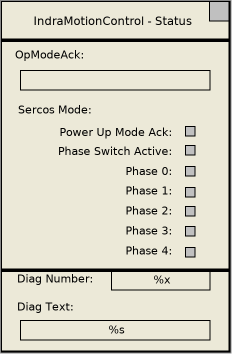
VISUALIZATION ImcStatus  // 232x354
    Rectangle (0,0 230x352)
    Rectangle (13,11 200x20), "IndraMotionControl - Status"
    Rectangle (209,1 20x20), colour toggle: Global_ImcInterface.ImcStatus .InOperation
    Rectangle (12,45 96x20), "OpModeAck:"
    Rectangle (20,70 190x20), text list: 'ImcModeStatus', text index: Global_ImcInterface.ImcStatus .Admin._OpModeAck
    Rectangle (0,40 230x0)
    Rectangle (15,100 90x20), "Sercos Mode:"
    Rectangle (0,270 230x0)
    Rectangle (185,187 10x10), colour toggle: Global_ImcInterface.ImcStatus .Admin.ModeStatus_P1
    Rectangle (185,226 10x10), colour toggle: Global_ImcInterface.ImcStatus .Admin.ModeStatus_P3
    Rectangle (185,206 10x10), colour toggle: Global_ImcInterface.ImcStatus .Admin.ModeStatus_P2
    Rectangle (185,166 10x10), colour toggle: Global_ImcInterface.ImcStatus .Admin.ModeStatus_P0
    Rectangle (185,247 10x10), colour toggle: Global_ImcInterface.ImcStatus .Admin.ModeStatus_BB
    Rectangle (185,145 10x10), colour toggle: Global_ImcInterface.ImcStatus .Admin.PhaseSwitchActive
    Rectangle (115,161 60x21), "Phase 0:"
    Rectangle (115,181 60x20), "Phase 1:"
    Rectangle (115,201 60x20), "Phase 2:"
    Rectangle (115,221 60x20), "Phase 3:"
    Rectangle (115,241 60x20), "Phase 4:"
    Rectangle (45,141 130x21), "Phase Switch Active:"
    Rectangle (45,125 130x15), "Power Up Mode Ack:"
    Rectangle (185,126 10x10), colour toggle: Global_ImcInterface.ImcStatus .Admin.PwrUpModeAck
    Rectangle (111,270 99x20), "%x", text variable: Global_ImcInterface.ImcStatus .Diag.Number
    Rectangle (20,320 190x20), "%s", text variable: Global_ImcInterface.ImcStatus .Diag.Message
    Rectangle (14,269 100x20), "Diag Number:"
    Rectangle (14,297 100x20), "Diag Text:"
END_VISUALIZATION

// IndraMotionMlc1/Application/AxisInterface/Visualizations/SystemOverview/System_Overview
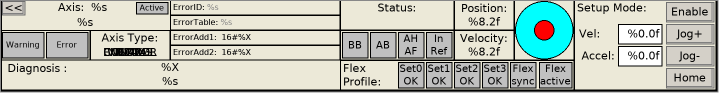
VISUALIZATION System_Overview  // 719x93
VAR_INPUT
	m_Input_AxisName : AXIS_REF;
END_VAR
    Rectangle (0,-1 717x92)
    Rectangle (1,61 340x15), "Diagnosis :"
    Rectangle (0,30 90x30)
    Rectangle (0,15 170x15), "%s", text variable: arAxisStatus_gb[m_Input_AxisName.AxisNo].Admin.Name
    Rectangle (340,30 114x30)
    Rectangle (514,0 60x60)
    Rectangle (24,0 117x15), "Axis: %s", text variable: m_Input_AxisName.AxisNo
    Rectangle (340,0 114x30), "Status:"
    Rectangle (454,0 60x30), "Position: %8.2f", text variable: AxisData[m_Input_AxisName.AxisNo].rActualPosition_i
    Rectangle (454,30 60x30), "Velocity: %8.2f", text variable: AxisData[m_Input_AxisName.AxisNo].rActualVelocity_i
    RoundedRectangle (342,32 26x26), "BB", colour toggle: (AxisData[m_Input_AxisName.Axisno].Axis_Inbb) <> 0
    RoundedRectangle (370,32 26x26), "AB", colour toggle: (AxisData[m_Input_AxisName.Axisno].Axis_InAb) <> 0
    RoundedRectangle (426,32 26x26), "In Ref", colour toggle: (AxisData[m_Input_AxisName.Axisno].Axis_Homed) <> 0
    RoundedRectangle (2,32 42x26), "Warning", colour toggle: (arAxisStatus_gb[m_Input_AxisName.Axisno].Diag.Warning) <> 0
    RoundedRectangle (46,32 42x26), "Error", colour toggle: (arAxisStatus_gb[m_Input_AxisName.Axisno].Diag.Error) <> 0
    RoundedRectangle (398,32 26x26), "AH AF", colour toggle: (AxisData[m_Input_AxisName.Axisno].Axis_Power) <> 0
    Ellipse (515,1 58x58)
    Polygon (0,0 0x0)
        p2858320360: AxisData[m_Input_AxisName.Axisno].rActualPosition_i
    Ellipse (534,20 20x20), colour toggle: (arAxisStatus_gb[m_Input_AxisName.AxisNo].Admin.Active) <> 0
    Rectangle (90,30 80x30), "Axis Type:"
    Rectangle (574,0 143x90), "Setup Mode:"
    Button (666,2 48x20), "Enable", colour toggle: arAxisStatus_gb[m_Input_AxisName.AxisNo].SetupMode.EnableAck, pressed state: arAxisCtrl_gb [m_Input_AxisName.AxisNo].SetupMode.Enable, input disabled if: bRemoteOn_gb = FALSE
        toggle arAxisCtrl_gb [m_Input_AxisName.AxisNo].SetupMode.Enable
    Button (666,24 48x20), "Jog+", input disabled if: (arAxisStatus_gb[m_Input_AxisName.AxisNo].SetupMode.EnableAck) = 0
        tap arAxisCtrl_gb [m_Input_AxisName.AxisNo].SetupMode.JogPlus
    Button (666,46 48x20), "Jog-", input disabled if: (arAxisStatus_gb[m_Input_AxisName.AxisNo].SetupMode.EnableAck) = 0
        tap arAxisCtrl_gb [m_Input_AxisName.AxisNo].SetupMode.JogMinus
    Button (666,68 48x20), "Home", colour toggle: arAxisStatus_gb[m_Input_AxisName.AxisNo].SetupMode.HomingAck, input disabled if: (arAxisStatus_gb[m_Input_AxisName.AxisNo].SetupMode.EnableAck) = 0
        tap arAxisCtrl_gb [m_Input_AxisName.AxisNo].SetupMode.Homing
    Rectangle (618,24 44x20), "%0.0f", text variable: arAxisCtrl_gb[m_Input_AxisName.AxisNo].SetupMode.Vel
        OnMouseUp: write arAxisCtrl_gb [m_Input_AxisName.AxisNo].SetupMode.Vel via Edit
    Rectangle (575,24 29x20), "Vel:"
    Rectangle (618,46 44x20), "%0.0f", text variable: arAxisCtrl_gb[m_Input_AxisName.AxisNo].SetupMode.Accel
        OnMouseUp: write arAxisCtrl_gb [m_Input_AxisName.AxisNo].SetupMode.Accel via Edit
    Rectangle (575,46 46x20), "Accel:"
    Button (2,1 23x14), "<<"
        OnMouseClick:  Assign=Axis_Overview, Type=Assignment
        OnMouseClick: execute { VisuAxisNo :=(m_Input_AxisName.AxisNo); }
    RoundedRectangle (136,2 32x12), "Active", colour toggle: (arAxisStatus_gb[m_Input_AxisName.AxisNo].Admin.Active) <> 0
    Rectangle (0,60 340x15), "%X", text variable: arAxisStatus_gb [m_Input_AxisName.AxisNo].Diag.Number, invisible if: arAxisStatus_gb [m_Input_AxisName.AxisNo].Diag.Number = 0
    RoundedRectangle (398,62 26x26), "Set0 OK", colour toggle: (AxisData[m_Input_AxisName.Axisno].FlexProfil_Set0_Ok) <> 0
    RoundedRectangle (426,62 26x26), "Set1 OK", colour toggle: (AxisData[m_Input_AxisName.Axisno].FlexProfil_Set1_Ok) <> 0
    RoundedRectangle (454,62 26x26), "Set2 OK", colour toggle: (AxisData[m_Input_AxisName.Axisno].FlexProfil_Set2_Ok) <> 0
    RoundedRectangle (482,62 26x26), "Set3 OK", colour toggle: (AxisData[m_Input_AxisName.Axisno].FlexProfil_Set3_Ok) <> 0
    Group (90,45 80x15)
        Rectangle (0,0 80x15), "REAL", invisible if: arAxisStatus_gb [m_Input_AxisName.AxisNo].Admin.AxisType <> RealAxisCfg
        Rectangle (0,0 80x15), "VIRTUAL", invisible if: arAxisStatus_gb [m_Input_AxisName.AxisNo].Admin.AxisType <> VirtualAxisCfg
        Rectangle (0,0 80x15), "ENCODER", invisible if: arAxisStatus_gb [m_Input_AxisName.AxisNo].Admin.AxisType <> EncoderAxisCfg
        Rectangle (0,0 80x15), "LINK", invisible if: arAxisStatus_gb [m_Input_AxisName.AxisNo].Admin.AxisType <> LinkAxisCfg
        Rectangle (0,0 80x15), "NO AXIS", invisible if: .arAxisStatus_gb [m_Input_AxisName.AxisNo].Admin.AxisType <> NoAxisConfig
        Rectangle (0,0 80x15), "CONTROL", invisible if: arAxisStatus_gb [m_Input_AxisName.AxisNo].Admin.AxisType <> ControlAxisCfg
    Rectangle (0,74 340x15), "%s", text variable: arAxisStatus_gb [m_Input_AxisName.AxisNo].Diag.Message
    Rectangle (170,0 170x15), "ErrorID: %s", text variable: arAxisStatus_gb [m_Input_AxisName.AxisNo].Diag.ErrorID, invisible if: (arAxisStatus_gb[m_Input_AxisName.Axisno].Diag.Error) <> 0
    Rectangle (170,0 170x15), "ErrorID:", invisible if: (arAxisStatus_gb[m_Input_AxisName.Axisno].Diag.Error) = 0, text list: 'ErrorIDCode', text index: arAxisStatus_gb [m_Input_AxisName.AxisNo].Diag.ErrorID
    Rectangle (170,15 170x15), "ErrorTable: %s", text variable: arAxisStatus_gb [m_Input_AxisName.AxisNo].Diag.ErrorIdent.Table, invisible if: (arAxisStatus_gb[m_Input_AxisName.Axisno].Diag.Error) <> 0
    Rectangle (170,15 170x15), "ErrorTable:", invisible if: (arAxisStatus_gb[m_Input_AxisName.Axisno].Diag.Error) = 0, text list: 'ErrorTable', text index: arAxisStatus_gb [m_Input_AxisName.AxisNo].Diag.ErrorIdent.Table
    Group (170,30 170x15)
        Rectangle (0,0 170x15), "ErrorAdd1: 16#%X", text variable: arAxisStatus_gb [m_Input_AxisName.AxisNo].Diag.ErrorIdent.Additional1, invisible if: (arAxisStatus_gb[m_Input_AxisName.Axisno].Diag.Error) <> 0
        Rectangle (0,0 170x15), "ErrorAdd1: 16#%X", text variable: arAxisStatus_gb [m_Input_AxisName.AxisNo].Diag.ErrorIdent.Additional1, invisible if: (arAxisStatus_gb[m_Input_AxisName.Axisno].Diag.Error) = 0
    Group (170,45 170x15)
        Rectangle (0,0 170x15), "ErrorAdd2: 16#%X", text variable: arAxisStatus_gb [m_Input_AxisName.AxisNo].Diag.ErrorIdent.Additional2, invisible if: (arAxisStatus_gb[m_Input_AxisName.Axisno].Diag.Error) <> 0
        Rectangle (0,0 170x15), "ErrorAdd2: 16#%X", text variable: arAxisStatus_gb [m_Input_AxisName.AxisNo].Diag.ErrorIdent.Additional2, invisible if: (arAxisStatus_gb[m_Input_AxisName.Axisno].Diag.Error) = 0
    Rectangle (340,60 234x30), "Flex Profile:"
    RoundedRectangle (539,62 33x26), "Flex active", colour toggle: (AxisData[m_Input_AxisName.Axisno].FlexProfil_Active) <> 0
    RoundedRectangle (510,62 26x26), "Flex sync", colour toggle: (AxisData[m_Input_AxisName.Axisno].FlexProfil_Sync) <> 0
    Rectangle (341,15 111x15), text list: 'AxisMode', text index: arAxisStatus_gb [m_Input_AxisName.AxisNo].Admin._OpModeAck
END_VISUALIZATION

// IndraMotionMlc1/Application/AxisInterface/Visualizations/SystemOverview/System_Overview_All_Axis
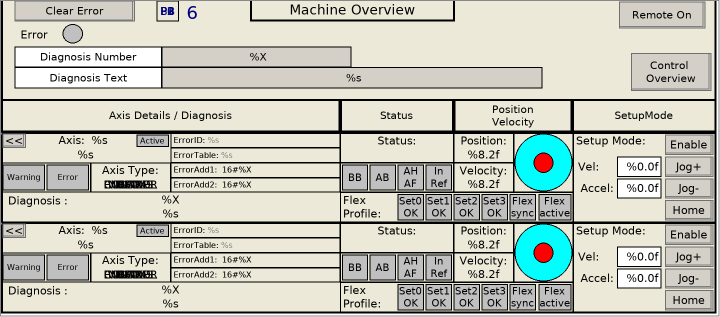
VISUALIZATION System_Overview_All_Axis  // 720x317
    Frame (1,-2 717x136)
        shows System_Overview_header()
    Frame (1,133 717x92)
        shows System_Overview(m_Input_AxisName := MyVirtualAxis1)
    Frame (1,223 717x92)
        shows System_Overview(m_Input_AxisName := MyVirtualAxis2)
END_VISUALIZATION

// IndraMotionMlc1/Application/AxisInterface/Visualizations/SystemOverview/System_Overview_header
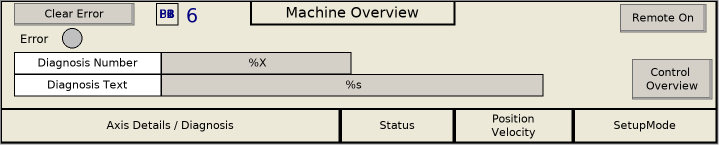
VISUALIZATION System_Overview_header  // 719x145
    Rectangle (0,0 717x143)
    Rectangle (340,108 114x35), "Status"
    Rectangle (0,108 340x35), "Axis Details / Diagnosis"
    Rectangle (454,108 119x35), "Position Velocity"
    Rectangle (573,108 144x35), "SetupMode"
    Ellipse (62,28 20x20), colour toggle: Global_ImcInterface.ImcStatus.Diag.Error
    Rectangle (17,29 50x20), "Error"
    Rectangle (250,0 205x25), "Machine Overview"
    Button (632,59 80x40), "Control Overview"
        OnMouseUp:  Assign=ImcInterface_Status_control, Assign=ImcInterface_Status_control, Type=Assignment
    Button (14,3 120x22), "Clear Error", input disabled if: bRemoteOn_gb = FALSE
        tap Global_ImcInterface.ImcCtrl .Admin.ClearError
    Rectangle (161,52 190x22), "%X", text variable: Global_ImcInterface.ImcStatus.Diag.Number
    Rectangle (14,52 147x22), "Diagnosis Number"
    Rectangle (14,74 147x22), "Diagnosis Text"
    Rectangle (161,74 382x22), "%s", text variable: Global_ImcInterface.ImcStatus.Diag.Message
    Rectangle (156,3 22x22), "P2", invisible if: NOT Global_ImcInterface.ImcStatus.Admin.ModeStatus_P2
    Rectangle (156,3 22x22), "BB", invisible if: NOT Global_ImcInterface.ImcStatus.Admin.ModeStatus_BB
    Rectangle (156,3 22x22), "P0", invisible if: NOT Global_ImcInterface.ImcStatus.Admin.ModeStatus_P0
    Rectangle (156,3 22x22), "P3", invisible if: NOT Global_ImcInterface.ImcStatus.Admin.ModeStatus_P3
    Rectangle (156,3 22x22), "P1", invisible if: NOT Global_ImcInterface.ImcStatus.Admin.ModeStatus_P1
    Rectangle (181,5 22x22), "6", invisible if: NOT Global_ImcInterface.ImcStatus.Admin.PhaseSwitchActive
    Button (620,4 86x28), "Remote On", colour toggle: UserVarGlobal.bRemoteOn_gb
        toggle UserVarGlobal.bRemoteOn_gb
END_VISUALIZATION

// IndraMotionMlc1/Application/AxisInterface/Visualizations/Utilities/AdjustPosition
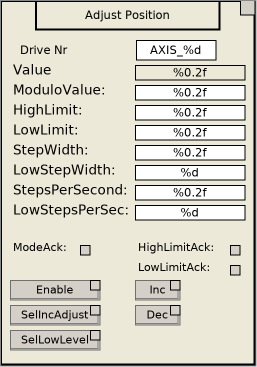
VISUALIZATION AdjustPosition  // 257x367
    Rectangle (0,0 255x365)
    Rectangle (35,0 185x30), "Adjust Position"
    Rectangle (10,80 118x20), "ModuloValue:"
    Rectangle (135,85 110x15), "%0.2f", text variable: arAxisCtrl_gb[VisuAxisNo].PosMode.Adjust.AdjModuloValue
        OnMouseUp: write the text variable via Edit
    Button (10,280 90x20), "Enable"
        OnMouseClick:  ToggleVariable=arAxisCtrl_gb[VisuAxisNo].PosMode.Adjust.Enable
    Rectangle (80,245 10x10), colour toggle: (arAxisStatus_gb[VisuAxisNo].PosMode.Adjust.ModeAck) <> 0
    Rectangle (10,100 90x20), "HighLimit:"
    Rectangle (135,105 110x15), "%0.2f", text variable: arAxisCtrl_gb[VisuAxisNo ].PosMode.Adjust.HighLimit
        OnMouseUp: write the text variable via Edit
    Rectangle (10,120 90x20), "LowLimit:"
    Rectangle (135,125 110x15), "%0.2f", text variable: arAxisCtrl_gb[VisuAxisNo].PosMode.Adjust.LowLimit
        OnMouseUp: write the text variable via Edit
    Rectangle (10,140 90x20), "StepWidth:"
    Rectangle (135,145 110x15), "%0.2f", text variable: arAxisCtrl_gb[VisuAxisNo].PosMode.Adjust.StepWidth
        OnMouseUp: write the text variable via Edit
    Rectangle (10,160 128x20), "LowStepWidth:"
    Rectangle (135,165 110x15), "%d", text variable: arAxisCtrl_gb[VisuAxisNo].PosMode.Adjust.LowStepWidth
        OnMouseUp: write the text variable via Edit
    Rectangle (10,180 148x20), "StepsPerSecond:"
    Rectangle (135,185 110x15), "%0.2f", text variable: arAxisCtrl_gb[VisuAxisNo].PosMode.Adjust.StepsPerSecond
        OnMouseUp: write the text variable via Edit
    Rectangle (10,200 148x20), "LowStepsPerSec:"
    Rectangle (135,205 110x15), "%d", text variable: arAxisCtrl_gb[VisuAxisNo].PosMode.Adjust.LowStepsPerSec
        OnMouseUp: write the text variable via Edit
    Rectangle (135,260 90x15), "LowLimitAck:"
    Rectangle (230,245 10x10), colour toggle: (arAxisStatus_gb[VisuAxisNo].PosMode.Adjust.HighLimitAck) <> 0
    Rectangle (135,240 90x15), "HighLimitAck:"
    Rectangle (230,265 10x10), colour toggle: (arAxisStatus_gb[VisuAxisNo].PosMode.Adjust.LowLimitAck) <> 0
    Button (10,305 90x20), "SelIncAdjust"
        OnMouseClick:  ToggleVariable=arAxisCtrl_gb[VisuAxisNo].PosMode.Adjust.SelIncAdjust
    Button (135,280 45x20), "Inc"
        OnMouseDown:  ToggleVariable=arAxisCtrl_gb[VisuAxisNo].PosMode.Adjust.Inc
        OnMouseUp:  ToggleVariable=arAxisCtrl_gb[VisuAxisNo].PosMode.Adjust.Inc
    Button (135,305 45x20), "Dec"
        OnMouseDown:  ToggleVariable=arAxisCtrl_gb[VisuAxisNo].PosMode.Adjust.Dec
        OnMouseUp:  ToggleVariable=arAxisCtrl_gb[VisuAxisNo].PosMode.Adjust.Dec
    Button (10,330 90x20), "SelLowLevel"
        OnMouseClick:  ToggleVariable=arAxisCtrl_gb[VisuAxisNo].PosMode.Adjust.SelLowLevel
    Rectangle (10,240 65x15), "ModeAck:"
    Rectangle (90,280 10x10), colour toggle: (arAxisCtrl_gb[VisuAxisNo].PosMode.Adjust.Enable) <> 0
    Rectangle (170,280 10x10), colour toggle: (arAxisCtrl_gb[VisuAxisNo].PosMode.Adjust.Inc) <> 0
    Rectangle (170,305 10x10), colour toggle: (arAxisCtrl_gb[VisuAxisNo].PosMode.Adjust.Dec) <> 0
    Rectangle (90,305 10x10), colour toggle: (arAxisCtrl_gb[VisuAxisNo].PosMode.Adjust.SelIncAdjust) <> 0
    Rectangle (90,330 10x10), colour toggle: (arAxisCtrl_gb[VisuAxisNo].PosMode.Adjust.SelLowLevel) <> 0
    Rectangle (135,65 110x15), "%0.2f", text variable: arAxisCtrl_gb[VisuAxisNo ].PosMode.Position
    Rectangle (240,0 15x15), colour toggle: (arAxisStatus_gb[VisuAxisNo].Admin._OpModeAck) = ModePosAbs
    Rectangle (10,60 118x20), "Value"
    Rectangle (0,40 70x20), "Drive Nr"
    Rectangle (136,40 80x20), "AXIS_%d", text variable: VisuAxisNo
        OnMouseUp: write the text variable via Edit
END_VISUALIZATION

// IndraMotionMlc1/Application/AxisInterface/Visualizations/Utilities/AdjustVelocity
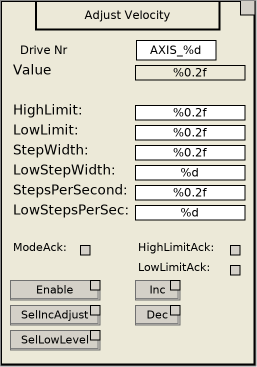
VISUALIZATION AdjustVelocity  // 257x367
    Rectangle (0,0 255x365)
    Rectangle (35,0 185x30), "Adjust Velocity"
    Button (10,280 90x20), "Enable"
        OnMouseClick:  ToggleVariable=arAxisCtrl_gb[VisuAxisNo].VelMode.Adjust.Enable
    Rectangle (80,245 10x10), colour toggle: (arAxisStatus_gb[VisuAxisNo].VelMode.Adjust.ModeAck) <> 0
    Rectangle (10,100 90x20), "HighLimit:"
    Rectangle (135,105 110x15), "%0.2f", text variable: arAxisCtrl_gb[VisuAxisNo ].VelMode.Adjust.HighLimit
        OnMouseUp: write the text variable via Edit
    Rectangle (10,120 90x20), "LowLimit:"
    Rectangle (135,125 110x15), "%0.2f", text variable: arAxisCtrl_gb[VisuAxisNo].VelMode.Adjust.LowLimit
        OnMouseUp: write the text variable via Edit
    Rectangle (10,140 90x20), "StepWidth:"
    Rectangle (135,145 110x15), "%0.2f", text variable: arAxisCtrl_gb[VisuAxisNo].VelMode.Adjust.StepWidth
        OnMouseUp: write the text variable via Edit
    Rectangle (10,160 128x20), "LowStepWidth:"
    Rectangle (135,165 110x15), "%d", text variable: arAxisCtrl_gb[VisuAxisNo].VelMode.Adjust.LowStepWidth
        OnMouseUp: write the text variable via Edit
    Rectangle (10,180 148x20), "StepsPerSecond:"
    Rectangle (135,185 110x15), "%0.2f", text variable: arAxisCtrl_gb[VisuAxisNo].VelMode.Adjust.StepsPerSecond
        OnMouseUp: write the text variable via Edit
    Rectangle (10,200 148x20), "LowStepsPerSec:"
    Rectangle (135,205 110x15), "%d", text variable: arAxisCtrl_gb[VisuAxisNo].VelMode.Adjust.LowStepsPerSec
        OnMouseUp: write the text variable via Edit
    Rectangle (135,260 90x15), "LowLimitAck:"
    Rectangle (230,245 10x10), colour toggle: (arAxisStatus_gb[VisuAxisNo].VelMode.Adjust.HighLimitAck) <> 0
    Rectangle (135,240 90x15), "HighLimitAck:"
    Rectangle (230,265 10x10), colour toggle: (arAxisStatus_gb[VisuAxisNo].VelMode.Adjust.LowLimitAck) <> 0
    Button (10,305 90x20), "SelIncAdjust"
        OnMouseClick:  ToggleVariable=arAxisCtrl_gb[VisuAxisNo].VelMode.Adjust.SelIncAdjust
    Button (135,280 45x20), "Inc"
        OnMouseDown:  ToggleVariable=arAxisCtrl_gb[VisuAxisNo].VelMode.Adjust.Inc
        OnMouseUp:  ToggleVariable=arAxisCtrl_gb[VisuAxisNo].VelMode.Adjust.Inc
    Button (135,305 45x20), "Dec"
        OnMouseDown:  ToggleVariable=arAxisCtrl_gb[VisuAxisNo].VelMode.Adjust.Dec
        OnMouseUp:  ToggleVariable=arAxisCtrl_gb[VisuAxisNo].VelMode.Adjust.Dec
    Button (10,330 90x20), "SelLowLevel"
        OnMouseClick:  ToggleVariable=arAxisCtrl_gb[VisuAxisNo].VelMode.Adjust.SelLowLevel
    Rectangle (10,240 65x15), "ModeAck:"
    Rectangle (90,280 10x10), colour toggle: (arAxisCtrl_gb[VisuAxisNo].VelMode.Adjust.Enable) <> 0
    Rectangle (170,280 10x10), colour toggle: (arAxisCtrl_gb[VisuAxisNo].VelMode.Adjust.Inc) <> 0
    Rectangle (170,305 10x10), colour toggle: (arAxisCtrl_gb[VisuAxisNo].VelMode.Adjust.Dec) <> 0
    Rectangle (90,305 10x10), colour toggle: (arAxisCtrl_gb[VisuAxisNo].VelMode.Adjust.SelIncAdjust) <> 0
    Rectangle (90,330 10x10), colour toggle: (arAxisCtrl_gb[VisuAxisNo].VelMode.Adjust.SelLowLevel) <> 0
    Rectangle (135,65 110x15), "%0.2f", text variable: arAxisCtrl_gb[VisuAxisNo ].VelMode.Velocity
    Rectangle (240,0 15x15), colour toggle: (arAxisStatus_gb[VisuAxisNo].Admin._OpModeAck) = ModeVel
    Rectangle (10,60 118x20), "Value"
    Rectangle (0,40 70x20), "Drive Nr"
    Rectangle (136,40 80x20), "AXIS_%d", text variable: VisuAxisNo
        OnMouseUp: write the text variable via Edit
END_VISUALIZATION

(* text list AxisMode (id | default)
  0 | ModeAB
  1 | ModeAH
  2 | ModeHoming
  4 | ModePosAbs
  8 | ModePosRel
  16 | ModePosAdd
  32 | ModeVel
  64 | ModeSyncPhase
  128 | ModeSyncVel
  256 | ModeSyncCam
  512 | ModeSyncProfile
  1024 | ModeTorque
  2048 | ModeFlexProfile
  4096 | ModeStopping
  8192 | ModeCoordinated
  16384 | ModeInterrupted
  32768 | ModeExternalFB
  65536 | ModeCyclicPos
  131072 | ModeCyclicVel
  262144 | ModeCyclicTrq
  524288 | ModeXx_User_1
  1048576 | ModeXx_User_2
  2097152 | ModeXx_User_3
  4194304 | ModeXx_User_4
  8388608 | ModeXx_User_5
  16777216 | ModeXx_User_6
  33554432 | ModeXx_User_7
  67108864 | ModeXx_User_8
  134217728 | ModePosAbs2
  268435456 | ModeValveCtrl
   |  *)

(* text list ExecutionMode (id | default)
  0 | EXECUTE_CYCLIC
  1 | EXECUTE_SINGLE
   |  *)

(* text list ProfileEntry (id | default)
  0 | SLAVE_ORIGIN_MASTER_ORIGIN
  1 | SLAVE_CURRENT_MASTER_CURRENT
  2 | SLAVE_ORIGIN_MASTER_CURRENT
  3 | SLAVE_CURRENT_MASTER_ORIGIN
  4 | SLAVE_RELATIVE_MASTER_ORIGIN
   |  *)

(* text list StartMode (id | default)
  0 | ABSOLUTE
  1 | RELATIVE
  2 | ABSOLUTE_RAMPIN
  3 | RELATIVE_RAMPIN
   |  *)

(* text list SyncDirection (id | default)
  0 | SHORTEST_WAY
  1 | CATCH_UP
  2 | SLOW_DOWN
   |  *)

(* text list SyncType (id | default)
  0 | SYNC_RAMPIN_SHORTEST_WAY
  1 | SYNC_RAMPIN_CATCH_UP
  2 | SYNC_RAMPIN_SLOW_DOWN
  3 | SYNC_DIRECT
   |  *)

(* text list ImcModeControl (id | default)
  0 | IMC_MODE_CTRL_P0
  2 | IMC_MODE_CTRL_P2
  4 | IMC_MODE_CTRL_BB
   |  *)

(* text list ImcModeStatus (id | default)
  0 | IMC_MODE_STATUS_P0
  1 | IMC_MODE_STATUS_P1
  2 | IMC_MODE_STATUS_P2
  3 | IMC_MODE_STATUS_P3
  4 | IMC_MODE_STATUS_BB
  255 | IMC_MODE_UNDEFINED
   |  *)

(* text list ErrorIDCode (id | default)
  0 | NONE_ERROR
  1 | INPUT_INVALID_ERROR
  2 | COMMUNICATION_ERROR
  3 | RESOURCE_ERROR
  4 | ACCESS_ERROR
  5 | STATE_MACHINE_ERROR
  6 | INPUT_RANGE_ERROR
  7 | CALCULATION_ERROR
  8 | DEVICE_ERROR
  32766 | OTHER_ERROR
  32767 | SYSTEM_ERROR
   |  *)

(* text list ErrorTable (id | default)
  0 | NO_TABLE_USED
  16 | SERCOS_TABLE
  32 | MLD_TABLE
  48 | MLC_TABLE
  64 | MTX_TABLE
  80 | MLP_TABLE
  96 | PLC_TABLE
  112 | INDRV_TABLE
  128 | DIAX_TABLE
  144 | ECO_TABLE
  304 | PB_DP_TABLE
  320 | DEVICENET_TABLE
  336 | ETHERNET_TABLE
  337 | ETHERNET_IP_TABLE
  352 | INTERBUS_TABLE
  368 | F_RELATED_TABLE
  384 | CAN_TABLE
  400 | INLINEIO_TABLE
  512 | PROFINETIO_TABLE
  528 | S20_IO_TABLE
  544 | S67_IO_TABLE
  4096 | USER1_TABLE
  4097 | USER2_TABLE
  4098 | USER3_TABLE
  4099 | USER4_TABLE
  4100 | USER5_TABLE
  4101 | USER6_TABLE
  4102 | USER7_TABLE
  4103 | USER8_TABLE
  4104 | USER9_TABLE
  4105 | USER10_TABLE
   |  *)
